Staubli VAL3: selectNewField.pgx

public program selectNewField(screen& x_scr, num x_nSelected, num x_nIndex, num x_nView)
  local num l_nFirst
begin
  //-----------------------------------------------------------------------
  //Header begin
  //Description of program
  //  Select a new item with a user friendly system.
  //  Usually use when you create a new Item and you want to select it.
  //  This program update the list with the the element x_nSelected
  //  that you want to selected.
  //  选择与用户交互性友好系统的一个新条目
  //  当你去创建一个新条目，你想去选择它时，常常会使用
  //  该程序更新了你想去选择的元素x_nSelected列表。
  //Input parameters  输入参数
  //  num x_nSelected : 数值量x_nSelected
  //    role : position that you want to go in the list
  //    作用：你想去到的列表的位置
  //    possible values : - "-1" : place current selected element in the
  //    middle of the list.
  //                      - other values : place the element in the middle of the list.
  //    有可能的值：- "-1" ：放置目前已选的元素在列表的中部。
  //  num x_nIndex :
  //    role : current position in the list
  //    作用：列表中目前位置
  //  num x_nView :
  //    role : current position of the list cursor
  //    作用：列表光标目前的位置
  //Examples
  //  call selectNewField(scrMy,7,4,3)  //Displays the Item number 7 in the
  //                              middle of the list
  //  call selectNewField(scrMy,-1,7,4) //Place the current selected Item
  //                              in the middle of the list
  //
  //History
  //  Creation : 28-04-08 - f.Rob
  //
  //  Modified : 08-08-22 - J.Cook     Add screen parameter
  //Header end
  //-----------------------------------------------------------------------
  // Update the first value from the parameter
  l_nFirst=max(x_nIndex-x_nView,0)
  // Do only an update of the first item
  if (x_nSelected==-1)
    nView=x_nView
    call listUpdate(x_scr, x_nIndex-x_nView)
  else
    //Select the new field using a scroll logic
    //The new value is not in the screen
    if x_nSelected<l_nFirst or abs(x_nSelected-l_nFirst)>=(nBottomY)
      //Start from the beginnnig
      if x_nSelected<l_nFirst and x_nSelected<nBottomY
        nView=x_nSelected
        call listUpdate(x_scr, 0)
      else
        if x_nSelected<size(sItems)-nBottomY
          //Move the list and select the field in the middle
          nView=roundUp(nBottomY/2)
        else
          nView=x_nSelected-(size(sItems)-nBottomY)
        endIf
        call listUpdate(x_scr, abs(x_nSelected-nView))
      endIf
    else
      //Move only the nView of the field
      nView=abs(x_nSelected-l_nFirst)
      call listUpdate(x_scr, abs(x_nIndex-x_nView))
    endIf
  endIf
end
